PROGRAM MAIN
VAR
END_VAR

RunGrindingWell();

END_PROGRAM

(* stored: Version 1.1.0.1, ProductVersion 3.1.4024.4
   POU MAIN: Id {a4b3803a-ed89-49a3-96a7-2a90aa0e77b8}, SpecialFunc None *)
